{attribute 'qualified_only'}
VAR_GLOBAL
END_VAR

(* stored: Version 1.1.0.1, ProductVersion 3.1.4022.18
   GVL GVL_Motion: Id {18d82037-8457-400f-b1ad-ea349db133b4} *)
